{attribute 'qualified_only'}
VAR_GLOBAL
    (*******************************************************************)
    (* Allgemeine Globale Variablen *)
    (*******************************************************************)
    (******* FREIGABEN *********)
    //ST01
    xFG_ST01akVZ : BOOL; // Vereinzelung Teil anwesend
    xFG_ST01akWT : BOOL; // WT anwesend
    //ST02
    xFG_ST02akWT : BOOL; // WT anwesend

END_VAR

(* stored: Version 1.1.0.1, ProductVersion 3.1.4024.12
   GVL GVL: Id {94734850-411d-4576-a0e7-f0a38cdbbc44} *)
